// TIA Portal V18 export
VAR_GLOBAL   // PLC tag table "PLCIO_DI"
   "iHMI Control On" AT %I100.0 : Bool;   // HMI_上电按钮 / HMI_Power on button
   "iHMI Machine Start" AT %I100.1 : Bool;   // HMI_设备启动按钮 / HMI_Device start button
   "iHMI Machine Stop" AT %I100.2 : Bool;   // HMI_设备停止按钮 / HMI_Device Stop Button
   "iHMI ResetButton" AT %I100.3 : Bool;   // HMI_复位按钮 / HMI_reset button
   "iHMI Manual/Auto" AT %I100.4 : Bool;   // HMI_手/自动切换按钮 / HMI_Hand/auto switch button
   "iHMI Safety Gate Unlock" AT %I100.5 : Bool;   // HMI_安全门解锁按钮 / HMI_safety door unlock button
   "iHMI E-Stop" AT %I100.6 : Bool;   // HMI_急停 / HMI_Emergency stop
   "iRESERVE_I100.7" AT %I100.7 : Bool;   // 备用_I100.7 / Standby_I100.7
   iPressure AT %I101.0 : Bool;   // 气压监控 / Air pressure monitoring
   "iCircuit Breaker OK_1" AT %I101.1 : Bool;   // 电子断路器 OK_1 / Electronic circuit breaker OK_1
   "iCircuit Breaker OK_2" AT %I101.2 : Bool;   // 电子断路器 OK_2 / Electronic circuit breaker OK_2
   "iRESERVE_I101.3" AT %I101.3 : Bool;   // 备用_I101.3 / Standby_I101.3
   iE_StopButton2_A01 AT %I101.4 : Bool;   // A01急停按钮2 / A01 emergency stop button 2
   iNG_Button1 AT %I101.5 : Bool;   // NG下料按钮1 / NG blanking button 1
   iE_StopButton3_A02 AT %I101.6 : Bool;   // A02急停按钮3 / A02 emergency stop button 3
   iNG_Button2 AT %I101.7 : Bool;   // NG下料按钮2 / NG blanking button 2
   "iSafety door Locking FeedBack_1" AT %I102.0 : Bool;   // 安全门锁定反馈_1 / Safety door lock feedback_1
   "iSafety door Locking FeedBack_2" AT %I102.1 : Bool;   // 安全门锁定反馈_2 / Safety door lock feedback_2
   "iSafety door Locking FeedBack_3" AT %I102.2 : Bool;   // 安全门锁定反馈_3 / Safety door lock feedback_3
   "iSafety door Locking FeedBack_4" AT %I102.3 : Bool;   // 安全门锁定反馈_4 / Safety door lock feedback_4
   "iSafety door Locking FeedBack_5" AT %I102.4 : Bool;   // 安全门锁定反馈_5 / Safety door lock feedback_5
   "iSafety door Locking FeedBack_6" AT %I102.5 : Bool;   // 安全门锁定反馈_6 / Safety door lock feedback_6
   "iSafety door Locking FeedBack_7" AT %I102.6 : Bool;   // 安全门锁定反馈_7 / Safety door lock feedback_7
   "iSafety door Locking FeedBack_8" AT %I102.7 : Bool;   // 安全门锁定反馈_8 / Safety door lock feedback_8
   "iSafety Door Locking FeedBack" AT %I103.0 : Bool;   // 连锁安全门锁定反馈 / Interlocking security door lock feedback
   "iMateriel Door Locking FeedBack_H1" AT %I103.1 : Bool;   // 物料门锁定反馈_1 / Material door lock feedback_1
   "iMateriel Door Locking FeedBack_H2" AT %I103.2 : Bool;   // 物料门锁定反馈_2 / Material door lock feedback_2
   "iMateriel Door Locking FeedBack_J1" AT %I103.3 : Bool;   // 物料门锁定反馈_3 / Material door lock feedback_3
   "iMateriel Door Locking FeedBack_J2" AT %I103.4 : Bool;   // 物料门锁定反馈_4 / Material door lock feedback_4
   "iMateriel Door Locking FeedBack_K1" AT %I103.5 : Bool;   // 物料门锁定反馈_5 / Material door lock feedback_5
   "iMateriel Door Locking FeedBack_K2" AT %I103.6 : Bool;   // 物料门锁定反馈_6 / Material door lock feedback_6
   "iMateriel Door Locking FeedBack_L1" AT %I103.7 : Bool;   // 物料门锁定反馈_7 / Material door lock feedback_7
   iShaft_Button AT %I104.1 : Bool;   // shaft 上料按钮 / shaft loading button
   iE_StopButton4_H AT %I104.0 : Bool;   // H_急停按钮4 / H_Emergency stop button 4
   iShaft_EmptyButton AT %I104.2 : Bool;   // shaft 取空料盘按钮 / shaft empty tray button
   iE_StopButton5_J AT %I104.3 : Bool;   // J_急停按钮5 / J_Emergency stop button 5
   iMagnet_Button AT %I104.4 : Bool;   // Magnet上料按钮 / Magnet loading button
   iMagnet_EmptyButton AT %I104.5 : Bool;   // Magnet取空料盘按钮 / Magnet empty tray button
   iMagnet_UnlockButton AT %I104.6 : Bool;   // Magne门解锁按钮 / Magne door unlock button
   "iRESERVE_I104.7" AT %I104.7 : Bool;   // 备用_I104.7 / Standby_I104.7
   iE_StopButton6_K AT %I105.0 : Bool;   // K_急停按钮6 / K_Emergency stop button 6
   iReserved_Button AT %I105.1 : Bool;   // Reserved上料按钮 / Reserved feeding button
   iReserved_EmptyButton AT %I105.2 : Bool;   // Reserved取空料盘按钮 / Reserved empty tray button
   iReserved_UnlockButton AT %I105.3 : Bool;   // Reserved门解锁按钮 / Reserved door unlock button
   iE_StopButton7_L AT %I105.4 : Bool;   // L_急停按钮7 / L_Emergency stop button 7
   iUnloading_Button AT %I105.5 : Bool;   // Unloading按钮 / Unloading button
   iUnloading_EmptyButton AT %I105.6 : Bool;   // Unloading取空料盘按钮 / Unloading empty tray button
   iUnloading_UnlockButton AT %I105.7 : Bool;   // Unloading门解锁按钮 / Unloading door unlock button
   "iE-NG-01 Safety Gate_Open" AT %I106.0 : Bool;   // E-NG料盒-01安全门锁_a / E-NG material box-01 safety door lock_a
   "iE-NG-01 Safety Gate_UnLock" AT %I106.1 : Bool;   // E-NG料盒-01安全门锁_b / E-NG material box-01 safety door lock_b
   "iE-NG-02 Safety Gate_Open" AT %I106.2 : Bool;   // E-NG料盒-02安全门锁_a / E-NG material box-02 safety door lock_a
   "iE-NG-02 Safety Gate_UnLock" AT %I106.3 : Bool;   // E-NG料盒-02安全门锁_b / E-NG material box-02 safety door lock_b
   iALightCurtain_1 AT %I106.4 : Bool;   // 备用_I106.4 / A-Grating 1
   iALightCurtain_2 AT %I106.5 : Bool;   // 备用_I106.5 / A-Grating 2
   "iRESERVE_I106.6" AT %I106.6 : Bool;   // 备用_I106.6 / Standby_I106.6
   "iRESERVE_I106.7" AT %I106.7 : Bool;   // 备用_I106.7 / Standby_I106.7
   "iH-shaft Loading _a" AT %I107.0 : Bool;   // H-shaft上料线体驱动电机_a / H-shaft feeding line body drive motor_a
   "iH-shaft Loading _b" AT %I107.1 : Bool;   // H-shaft上料线体驱动电机_b / H-shaft feeding line body drive motor_b
   "iH-shaft Take _a" AT %I107.2 : Bool;   // H-shaft取空盘驱动电机_a / H-shaft takes empty plate drive motor_a
   "iH-shaft Take _b" AT %I107.3 : Bool;   // H-shaft取空盘驱动电机_b / H-shaft takes empty plate drive motor_b
   "iH-shaft  Lifting _a" AT %I107.4 : Bool;   // H-shaft 顶升位驱动电机_a / H-shaft lifting position drive motor_a
   "iH-shaft  Lifting _b" AT %I107.5 : Bool;   // H-shaft 顶升位驱动电机_b / H-shaft lifting position drive motor_b
   "iRESERVE_I107.6" AT %I107.6 : Bool;   // 备用_I107.6 / Standby_I107.6
   "iRESERVE_I107.7" AT %I107.7 : Bool;   // 备用_I107.7 / Standby_I107.7
   "iJ-magnet Loading _a" AT %I108.0 : Bool;   // J-magnet上料线体驱动电机_a / J-magnet loading wire body drive motor_a
   "iJ-magnet Loading _b" AT %I108.1 : Bool;   // J-magnet上料线体驱动电机_b / J-magnet feeding line body drive motor_b
   "iJ-magnet Take _a" AT %I108.2 : Bool;   // J-magnet取空盘驱动电机_a / J-magnet empty disk drive motor_a
   "iJ-magnet Take _b" AT %I108.3 : Bool;   // J-magnet取空盘驱动电机_b / J-magnet empty disk drive motor_b
   "iJ-magnet Lifting _a" AT %I108.4 : Bool;   // J-magnet顶升驱动电机_a / J-magnet jacking drive motor_a
   "iJ-magnet Lifting _b" AT %I108.5 : Bool;   // J-magnet顶升驱动电机_b / J-magnet jacking drive motor_b
   "iRESERVE_I108.6" AT %I108.6 : Bool;   // 备用_I108.6 / Standby_I108.6
   "iRESERVE_I108.7" AT %I108.7 : Bool;   // 备用_I108.7 / Standby_I108.7
   "iK-reserve Loading _a" AT %I109.0 : Bool;   // K-预留上料线体驱动电机_a / K-reserved feeding line body drive motor_a
   "iK-reserve Loading _b" AT %I109.1 : Bool;   // K-预留上料线体驱动电机_b / K-reserved feeding line body drive motor_b
   "iK-reserve Take _a" AT %I109.2 : Bool;   // K-预留取空盘驱动电机_a / K-reserved empty disk drive motor_a
   "iK-reserve Take _b" AT %I109.3 : Bool;   // K-预留取空盘驱动电机_b / K-reserved empty disk drive motor_b
   "iK-reserve Lifting3 _a" AT %I109.4 : Bool;   // K-预留顶升位3驱动电机_a / K-reserved lifting position 3 drive motor_a
   "iK-reserve Lifting3 _b" AT %I109.5 : Bool;   // K-预留顶升位3驱动电机_b / K-reserved lifting position 3 drive motor_b
   "iRESERVE_I109.6" AT %I109.6 : Bool;   // 备用_I109.6 / Standby_I109.6
   "iRESERVE_I109.7" AT %I109.7 : Bool;   // 备用_I109.7 / Standby_I109.7
   "iC- GluingDeviceReady" AT %I110.0 : Bool;   // C-涂胶模组点胶阀_a / C-gluing system ready
   "iC- GluingFault" AT %I110.1 : Bool;   // C-涂胶模组点胶阀_b / C-gluing system error
   "iC- GluingRefillTank" AT %I110.2 : Bool;   // C-涂胶模组点胶阀_c / C-glue coating system lacks material
   "iC- GluingTankEmpty" AT %I110.3 : Bool;   // 备用_I110.3 / C-glue coating system empty material
   "iL-Unloading Drive motor_a" AT %I110.4 : Bool;   // L-下料线体驱动电机_a / L-Blanking line drive motor_a
   "iL-Unloading Drive motor_b" AT %I110.5 : Bool;   // L-下料线体驱动电机_b / L-Blanking line drive motor_b
   "iL-Unloading transplanting motor_a" AT %I110.6 : Bool;   // L-下料线体移栽电机_a / L-Blanking wire body transplanting motor_a
   "iL-Unloading transplanting motor_b" AT %I110.7 : Bool;   // L-下料线体移栽电机_b / L-Blanking wire body transplanting motor_b
   iH_StopButton AT %I111.0 : Bool;
   iJ_StopButton AT %I111.1 : Bool;
   iK_StopButton AT %I111.2 : Bool;
   "iRESERVE_I111.3" AT %I111.3 : Bool;
   "iRESERVE_I111.4" AT %I111.4 : Bool;
   "iRESERVE_I111.5" AT %I111.5 : Bool;
   "iRESERVE_I111.6" AT %I111.6 : Bool;
   "iRESERVE_I111.7" AT %I111.7 : Bool;
END_VAR
